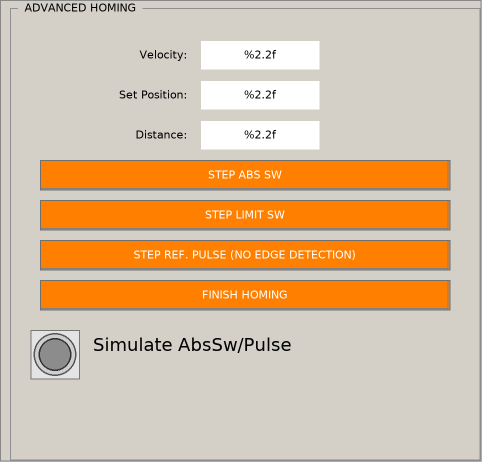
VISUALIZATION Homing  // 482x462
    GroupBox (10,0 470x460), "ADVANCED HOMING"
        Button (30,160 410x30), "STEP ABS SW"
            OnMouseClick: execute { GVL.axes[MAIN.hmiAxisSelect].eCommand:=eMcCommand.HomeStepAbsoluteSwitch; GVL.axes[MAIN.hmiAxisSelect].bEXECUTE:= TRUE; }
        Textfield (190,40 120x30), "%2.2f", text variable: GVL.axes[MAIN.hmiAxisSelect].fHomeVelocity
            OnMouseClick: write GVL.axes[MAIN.hmiAxisSelect].fHomeVelocity via Default
        Textfield (190,80 120x30), "%2.2f", text variable: GVL.axes[MAIN.hmiAxisSelect].fHomePosition
            OnMouseClick: write GVL.axes[MAIN.hmiAxisSelect].fHomePosition via Default
        Textfield (20,40 160x30), "Velocity:"
        Textfield (20,80 160x30), "Set Position:"
        Textfield (20,120 160x30), "Distance:"
        Button (30,280 410x30), "FINISH HOMING"
            OnMouseClick: execute { GVL.axes[MAIN.hmiAxisSelect].eCommand:=eMcCommand.HomeFinish; GVL.axes[MAIN.hmiAxisSelect].bEXECUTE:= TRUE; }
        PushSwitchLed (20,330 50x49), variable: GVL.axes[MAIN.hmiAxisSelect].MCSignalRef.Level, behaviour: TOGGLE, style: Switch-PushSwitchLed-Gray
        Button (30,200 410x30), "STEP LIMIT SW"
            OnMouseClick: execute { GVL.axes[MAIN.hmiAxisSelect].eCommand:=eMcCommand.HomeStepLimitSwitch; GVL.axes[MAIN.hmiAxisSelect].bEXECUTE:= TRUE; }
        Button (30,240 410x30), "STEP REF. PULSE (NO EDGE DETECTION)"
            OnMouseClick: execute { GVL.axes[MAIN.hmiAxisSelect].eCommand:=eMcCommand.HomeStepReferencePulse; GVL.axes[MAIN.hmiAxisSelect].bEXECUTE:= TRUE; }
    Textfield (200,120 120x30), "%2.2f", text variable: GVL.axes[MAIN.hmiAxisSelect].fHomeDistance
        OnMouseClick: write GVL.axes[MAIN.hmiAxisSelect].fHomeDistance via Default
    Label (90,330 280x30), "Simulate AbsSw/Pulse"
END_VISUALIZATION

(* stored: Version 1.1.0.1, ProductVersion 3.1.4022.12
   Visu Homing: Id {7a42f6ce-dc0c-4ea7-836d-e64c02cca468} *)
